GLOBALCONSTANTS DefaultPool (* Global constants *)
  PACKAGE Uebungen::const::UT::HystereseHorizontal;
  VAR_GLOBAL CONSTANT
    ISO_DESIGNATOR_WIDTH : UINT := 80;
    ISO_DESIGNATOR_HEIGHT : UINT := 80;
    ISO_MASK_SIZE : UINT := 480;
    ISO_VERSION_LABEL : STRING;
    MASK_WIDTH : UINT := 480;
    MASK_HEIGHT : UINT := 480;
    WorkingSet : UINT := 0;
    DataMask_M1 : UINT := 1000;
    Container_Schwellwerte : UINT := 3000;
    InputNumber_MID : UINT := 9000;
    InputNumber_DEAD : UINT := 9001;
    InputNumber_HYSTERESIS : UINT := 9002;
    OutputString_WorkingSet_0 : UINT := 11000;
    Polygon_MID : UINT := 16000;
    Polygon_MID_PLUS_DEAD : UINT := 16001;
    Polygon_MID_MINUS_DEAD : UINT := 16002;
    Polygon_MID_PLUS_DEAD_HYST : UINT := 16003;
    Polygon_MID_MINUS_DEAD_HYST : UINT := 16004;
    Bargraph_Hysterese : UINT := 18000;
    NumberVariable_MID : UINT := 21000;
    NumberVariable_DEAD : UINT := 21001;
    NumberVariable_HYSTERESIS : UINT := 21002;
    FontAttributes_6x8 : UINT := 23000;
    FontAttributes_Werte : UINT := 23001;
    LineStyle_Hysterese_MID_Gruen : UINT := 24000;
    LineStyle_Hysterese_DEAD_Orange : UINT := 24001;
    LineStyle_Hysterese_HYST_Rot : UINT := 24002;
    FillStyle_Hysterese_MID_Gruen : UINT := 25000;
    FillStyle_Hysterese_DEAD_Orange : UINT := 25001;
    FillStyle_Hysterese_HYST_Rot : UINT := 25002;
  END_VAR
END_GLOBALCONSTANTS
